PROGRAM Hardlopen
VAR
END_VAR

END_PROGRAM

(* stored: Version 1.1.0.1, ProductVersion 3.1.4024.15
   POU Hardlopen: Id {595a4fa8-c535-4084-8182-3622c9324e38}, SpecialFunc None *)
